(* Logix 5000 project; controller FRIST_EXAMPLE Emulate 5570 rev 19.11; software revision 19.01 *)

TASK MainTask (continuous, watchdog 500 ms) : MainProgram

MODULES
   Local : Emulate 5570 (ICP 2, rev 19.11)
       : 1756-IB32 (ICP 3, rev 3.1, Input RPI 20 ms)   // DG-INPUT
       : vendor 1 type 7 code 8 (ICP 4, rev 3.1, Output RPI 20 ms)
       : 1756-IF6I (ICP 5, rev 1.1, Input RPI 100 ms)
       : 1756-OF8 (ICP 6, rev 1.1, Output RPI 12 ms)
END_MODULES

VAR_GLOBAL   (* controller tags *)
   CMD_MT01 : BOOL;
   DESLIGA : BOOL := 1;
   LIGA : BOOL;
   PARAR : BOOL;
   REVERSO : BOOL;
   VAL_DIRETO : BOOL;
   VAL_REVERSO : BOOL;
END_VAR

PROGRAM MainProgram   (* main routine MainRoutine *)

ROUTINE MainRoutine   (* ladder *)
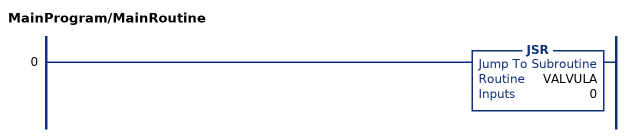
   0: JSR(VALVULA,0);
END_ROUTINE

ROUTINE VALVULA   (* ladder *)
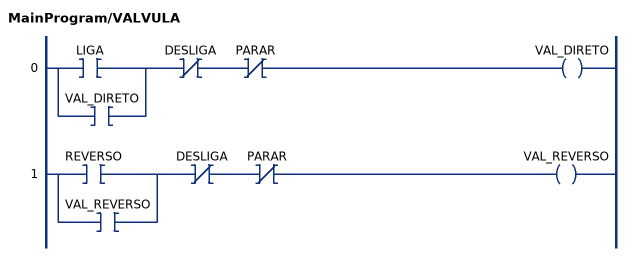
   0: [XIC(LIGA) ,XIC(VAL_DIRETO) ]XIO(DESLIGA)XIO(PARAR)OTE(VAL_DIRETO);
   1: [XIC(REVERSO) ,XIC(VAL_REVERSO) ]XIO(DESLIGA)XIO(PARAR)OTE(VAL_REVERSO);
END_ROUTINE
END_PROGRAM
